TYPE PositionRotations : 
STRUCT
	position : INT;
	rotations : INT;
END_STRUCT
END_TYPE

(* stored: Version 1.1.0.1, ProductVersion 3.1.4024.11
   DUT PositionRotations: Id {0867df64-b761-4321-a4de-cb69d48dd9cf} *)
